FUNCTION_BLOCK FB_ErrorState IMPLEMENTS I_State
VAR_INPUT
END_VAR
VAR_OUTPUT
END_VAR
VAR
	pMachine : POINTER TO FB_StateMachine;
END_VAR

PROPERTY Description : STRING
GET
Description := 'An error has occurred';
END_GET
END_PROPERTY

METHOD ErrorDetected : BOOL
VAR_IN_OUT
	errorEvents		: ST_ErrorEvents;
END_VAR
// transitionToErrorState(errorEvents := errorEvents, pMachine := pMachine);
END_METHOD

//FB_Init ist immer implizit verfügbar und wird primär für die Initialisierung verwendet.
//Der Rückgabewert wird nicht ausgewertet. Für gezielte Einflussnahme können Sie
//die Methoden explizit deklarieren und darin mit dem Standard-Initialisierungscode 
//zusätzlichen Code bereitstellen. Sie können den Rückgabewert auswerten.
METHOD FB_Init: BOOL
VAR_INPUT    
	bInitRetains: BOOL; // TRUE: Die Retain-Variablen werden initialisiert (Reset warm / Reset kalt)    
	bInCopyCode: BOOL;  // TRUE: Die Instanz wird danach in den Kopiercode kopiert (Online-Change)
	pMachine : POINTER TO FB_StateMachine;
END_VAR
THIS^.pMachine := pMachine;
END_METHOD

METHOD HeatIsRequested : BOOL
END_METHOD

PROPERTY Name : STRING
GET
Name := 'Error';
END_GET
END_PROPERTY

PROPERTY State : E_State
GET
State := E_State.ERROR;
END_GET
END_PROPERTY

METHOD TargetTemperatureReached : BOOL
END_METHOD

METHOD UserPressedConfirmationButton : BOOL
END_METHOD

METHOD UserPressedSwitchOffButton : BOOL
resetApplication(pMachine);
ADSLOGSTR(ADSLOG_MSGTYPE_HINT, 'Aus Button wurde gedrückt -> %s', pMachine^.OffState.Name);
pMachine^.SetState(pMachine^.OffState);
END_METHOD

METHOD UserPressedSwitchOnButton : BOOL
END_METHOD

METHOD WaterHasCooledDown : BOOL
END_METHOD

END_FUNCTION_BLOCK

(* stored: Version 1.1.0.1
   POU FB_ErrorState: Id {c6f603d6-7e40-4c21-bcd3-aae841f974cf}, SpecialFunc None
   Property Description: Id {99b20c4c-e12d-41aa-9edb-000ee4c7310b}
   Get Get: Id {22f33121-45f5-47c7-8aef-991291fe399a}
   Method ErrorDetected: Id {4858f92b-be7c-40d0-8ec0-7dce2aef6360}
   Method FB_init: Id {acff5f6f-b6a4-4746-b7e6-05f059e8448c}
   Method HeatIsRequested: Id {f5a49845-b3d2-4674-be77-835f5d419f38}
   Property Name: Id {cc46a02f-c560-4746-aafb-c4ebfec2dd31}
   Get Get: Id {e8bf7ff8-a2a9-4cce-99be-1ae11e37e3ab}
   Property State: Id {145413ed-c790-4267-82eb-9a9ffe70ba62}
   Get Get: Id {7228e2d1-54da-4346-af29-132743857a96}
   Method TargetTemperatureReached: Id {24b8b0f1-8ac1-4afc-bc6f-4eb4ccc3d660}
   Method UserPressedConfirmationButton: Id {3cfe4937-42e9-40a6-b5c7-527050ea73ed}
   Method UserPressedSwitchOffButton: Id {5bbcc8c1-3ef1-4641-89cd-a4c6e429c88b}
   Method UserPressedSwitchOnButton: Id {3b9616fd-86d5-4be9-a046-d7829150b454}
   Method WaterHasCooledDown: Id {3cab738b-672d-4222-9d6f-a0210fe54c6c} *)
